// TIA Portal V17 export
// export: Created 2022-05-07T16:38:48.5677688Z, ExportSetting WithDefaults, DisplayName Totally Integrated Automation Portal, DisplayVersion V17 Update 3, DisplayName TIA Portal Openness, DisplayVersion V17 Update 3, DisplayName TIA Portal Version Control Interface, DisplayVersion V17, DisplayName TIA Portal Test Suite Advanced, DisplayVersion V17 Update 1, DisplayName SINAMICS Startdrive Advanced, DisplayVersion V17 Update2, DisplayName SINAMICS Startdrive G130, G150, S120, S150, SINAMICS MV, S210, DisplayVersion V17 Update2, DisplayName SINAMICS Startdrive G110M, G120, G120C, G120D, G120P, G115D, DisplayVersion V17 Update2, DisplayName STEP 7 Professional, DisplayVersion V17 Update 3, DisplayName STEP 7 Safety, DisplayVersion V17, DisplayName WinCC UA Professional, DisplayVersion V17 Update 3
DATA_BLOCK "FB_ORG_ASSI_DB"   // DB13
VERSION : 0.1
// stored: AutoNumber true, DBAccessibleFromOPCUA true, InstanceOfName FB_ORG_ASSI, InstanceOfType FB
"FB_ORG_ASSI"
   // VAR
   //    CTRL_ASSE_STD_MA { S7_SetPoint := 'True'} : "CTRL_ASSE_STD";
   //    CTRL_ASSE_STD_MR { S7_SetPoint := 'True'} : "CTRL_ASSE_STD";
   //    CTRL_ASSE_STD_MS { S7_SetPoint := 'True'} : "CTRL_ASSE_STD";
   //    CTRL_ASSE_STD_ME { S7_SetPoint := 'True'} : "CTRL_ASSE_STD";
   // END_VAR
BEGIN
END_DATA_BLOCK
